FUNCTION F_USINT_RTN : USINT
VAR_INPUT
	stArg : ST_Arg;
END_VAR
VAR
	sysVar_Info : __SYSTEM.VAR_INFO;
END_VAR

sysVar_Info := __VARINFO(F_USINT_RTN);
IF stArg.TypeClass = sysVar_Info.TypeClass THEN 
	F_USINT_RTN := TO_USINT(stArg.sValue);
	END_IF

END_FUNCTION

(* stored: Version 1.1.0.1, ProductVersion 3.1.4024.4
   POU F_USINT_RTN: Id {e418ffc7-70d4-41a1-853c-bee74c274c68}, SpecialFunc None *)
